FUNCTION_BLOCK COMPARE_10593E80BE744DDAF (* Compare *)
  (* Standard: 61499-2 *)
  (* Version 1.0, 29.10.2008, marumil, nxtControl GmbH, Initial Version *)
  PACKAGE Main;
  (* Compiler Cpp *)
  {SET_ATTRIBUTE(Runtime.FBType.ImplementingType, Runtime.Standard#DYNGEN_COMPARE)}
  {SET_ATTRIBUTE(Configuration.GenericFBType.InterfaceParams, Runtime.Standard#CNT:=2;IN${CNT$}:STRING)}
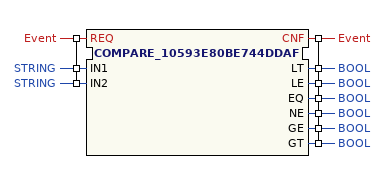
  EVENT_INPUT
    REQ WITH IN1, IN2; (* Normal Execution Request *)
  END_EVENT
  EVENT_OUTPUT
    CNF WITH LT, LE, EQ, NE, GE, GT; (* Execution Confirmation *)
  END_EVENT
  VAR_INPUT
    IN1 : STRING; (* Argument *)
    IN2 : STRING; (* Argument *)
  END_VAR
  VAR_OUTPUT
    LT : BOOL; (* IN1 < IN2 *)
    LE : BOOL; (* IN1 <= IN2 *)
    EQ : BOOL; (* IN1 = IN2 *)
    NE : BOOL; (* IN1 <> IN2 *)
    GE : BOOL; (* IN1 >= IN2 *)
    GT : BOOL; (* IN1 > IN2 *)
  END_VAR
  EC_STATES
    START;
  END_STATES
END_FUNCTION_BLOCK
